(* IEC 61131-3 sources: mastertool-rankine-bridge/tests/indexer/fixtures/sample_export/objects/application_fun_0__FunCalcularMedia, 2 files *)

(* ---- declaration.st ---- *)
FUNCTION FunCalcularMedia : REAL
VAR_INPUT
    rValorA         : REAL;
    rValorB         : REAL;
END_VAR
VAR
    rResultado      : REAL;
END_VAR

(* ---- implementation.st ---- *)
rResultado := (rValorA + rValorB) / 2;

IF rResultado > 100.0 THEN
    rResultado := 100.0;
ELSIF rResultado < 0.0 THEN
    rResultado := 0.0;
ELSE
    FbLimitador.Ajustar(
        IN_VALOR := rResultado,
        OUT_VALOR => rResultado
    );
END_IF;

FunCalcularMedia := rResultado;
